INTERFACE I_TempSensor EXTENDS I_ComponentBase

PROPERTY Temp : LREAL
GET
END_GET
END_PROPERTY

END_INTERFACE

(* stored: Version 1.1.0.1
   Itf I_TempSensor: Id {50c55809-fda1-447d-bc3e-8203634c9af0}
   Property Temp: Id {ce127390-c556-41bd-a4b2-3337fb4d92d9}
   Get Get: Id {80d78f06-89c8-4b0b-bd29-caf0d50c6508} *)
